FUNCTION_BLOCK FB_MotionVirtualFrame
(*
Takes 3 ST_MotionStages representing real axes that are orthogonal to each other and in a base frame of reference.
Takes 3 ST_MotionStages representing virtual axes that are orthogonal to each other and in a new frame of reference.
Computes the transformation from the base to the new frame of reference using 3 euler angles and a rotation order
as inputs. By default, the order and angles are interpreted as going from the base to the virtual frame. Can be
switched to go from virtual to base frame of reference.
If enabled, this function block will automatically handle commanding the real axes to move when the virtual axes
are commanded to move. If not enabled, the function block acts as a calculator, outputing the results of
calculating motions in a new frame of reference, but not changing any setpoints or commanding any moves.
*)
VAR_IN_OUT
    stMotionStageRx : ST_MotionStage; // Real X Axis in base frame of reference
    stMotionStageRy : ST_MotionStage; // Real Y Axis in base frame of reference
    stMotionStageRz : ST_MotionStage; // Real Z Axis in base frame of reference
    stMotionStageVx : ST_MotionStage; // Virtual X Axis in new frame of reference
    stMotionStageVy : ST_MotionStage; // Virtual Y Axis in new frame of reference
    stMotionStageVz : ST_MotionStage; // Virtual Z Axis in new frame of reference
END_VAR
VAR_INPUT
    (*TRUE to automatically overwrite real axis setpoints and command moves.
      FALSE to use this function only as a calculator.*)
    bEnable : BOOL;
    fAlphaDegrees : LREAL; // Angle of rotation about first axis.
    fBetaDegrees : LREAL; // Angle of rotation about second axis.
    fGammaDegrees : LREAL; // Angle of rotation about third axis.
    (*Rotation Order. E.g: XYZ to rotate alpha degrees around X axis, beta degrees around Y axis,
      and gamma degrees around Z axis. Valid rotation orders are:
      YZY, YXY, ZYZ, ZXZ, XYX, XZX, XYZ, YZX, ZXY, XZY, ZYX, YXZ.
      Default order for empty or invalid input is: ZYX.*)
    sOrder : STRING;
    (*FALSE to define inputs as rotating the frame of reference from the new frame to the base frame.
      TRUE to define the inputs as rotating the frame of reference from the base from to the new frame.*)
    bBaseToNew : BOOL := TRUE;
END_VAR
VAR_OUTPUT
    fbVirtActPositionVec3 : FB_Vec3;
    fbVirtActVelocityVec3 : FB_Vec3;
    fbVirtActAcceleraVec3 : FB_Vec3;

    fbRealTarPositionVec3 : FB_Vec3;
    fbRealTarVelocityVec3 : FB_Vec3;
    fbRealTarAcceleraVec3 : FB_Vec3;
END_VAR
VAR
    fAlphaRadians : LREAL;
    fBetaRadians : LREAL;
    fGammaRadians : LREAL;

    rtExecuteVx : R_TRIG;
    rtExecuteVy : R_TRIG;
    rtExecuteVz : R_TRIG;

    fbRealActPositionVec3 : FB_Vec3;
    fbRealActVelocityVec3 : FB_Vec3;
    fbRealActAcceleraVec3 : FB_Vec3;

    sOrderReversed : STRING;
    sLeft : STRING;
    sMid : STRING;
    sRight : STRING;

    fbVirtTarPositionVec3 : FB_Vec3;
    fbVirtTarVelocityVec3 : FB_Vec3;
    fbVirtTarAcceleraVec3 : FB_Vec3;
END_VAR


fAlphaRadians := DegToRad(fAlphaDegrees);
fBetaRadians := DegToRad(fBetaDegrees);
fGammaRadians := DegToRad(fGammaDegrees);

rtExecuteVx(CLK := stMotionStageVx.bExecute);
rtExecuteVy(CLK := stMotionStageVy.bExecute);
rtExecuteVz(CLK := stMotionStageVz.bExecute);

fbRealActPositionVec3.x := stMotionStageRx.Axis.NcToPlc.ActPos;
fbRealActPositionVec3.y := stMotionStageRy.Axis.NcToPlc.ActPos;
fbRealActPositionVec3.z := stMotionStageRz.Axis.NcToPlc.ActPos;

fbRealActVelocityVec3.x := stMotionStageRx.Axis.NcToPlc.ActVelo;
fbRealActVelocityVec3.y := stMotionStageRy.Axis.NcToPlc.ActVelo;
fbRealActVelocityVec3.z := stMotionStageRz.Axis.NcToPlc.ActVelo;

fbRealActAcceleraVec3.x := stMotionStageRx.Axis.NcToPlc.ActAcc;
fbRealActAcceleraVec3.y := stMotionStageRy.Axis.NcToPlc.ActAcc;
fbRealActAcceleraVec3.z := stMotionStageRz.Axis.NcToPlc.ActAcc;

sOrderReversed := ReverseOrder(sOrder);

IF bBaseToNew THEN
    RotatePosVelAccFrame(
        fbBaseFramePositionVec3 := fbRealActPositionVec3,
        fbBaseFrameVelocityVec3 := fbRealActVelocityVec3,
        fbBaseFrameAcceleraVec3 := fbRealActAcceleraVec3,
        fbNewFramePositionVec3 => fbVirtActPositionVec3,
        fbNewFrameVelocityVec3 => fbVirtActVelocityVec3,
        fbNewFrameAcceleraVec3 => fbVirtActAcceleraVec3,
        fAlphaRadians := fAlphaRadians,
        fBetaRadians := fBetaRadians,
        fGammaRadians := fGammaRadians,
        sOrder := sOrder
    );
ELSE
    RotatePosVelAccFrame(
        fbBaseFramePositionVec3 := fbRealActPositionVec3,
        fbBaseFrameVelocityVec3 := fbRealActVelocityVec3,
        fbBaseFrameAcceleraVec3 := fbRealActAcceleraVec3,
        fbNewFramePositionVec3 => fbVirtActPositionVec3,
        fbNewFrameVelocityVec3 => fbVirtActVelocityVec3,
        fbNewFrameAcceleraVec3 => fbVirtActAcceleraVec3,
        fAlphaRadians := -fGammaRadians,
        fBetaRadians := -fBetaRadians,
        fGammaRadians := -fAlphaRadians,
        sOrder := sOrderReversed
    );
END_IF

SetTargetPosVelAcc3D(
    stMotionStageX := stMotionStageVx,
    stMotionStageY := stMotionStageVy,
    stMotionStageZ := stMotionStageVz,
    fbActPosVec3 := fbVirtActPositionVec3,
    fbTarPosVec3 => fbVirtTarPositionVec3,
    fbTarVelVec3 => fbVirtTarVelocityVec3,
    fbTarAccVec3 => fbVirtTarAcceleraVec3
);

IF bBaseToNew THEN
    RotatePosVelAccFrame(
        fbBaseFramePositionVec3 := fbVirtTarPositionVec3,
        fbBaseFrameVelocityVec3 := fbVirtTarVelocityVec3,
        fbBaseFrameAcceleraVec3 := fbVirtTarAcceleraVec3,
        fbNewFramePositionVec3 => fbRealTarPositionVec3,
        fbNewFrameVelocityVec3 => fbRealTarVelocityVec3,
        fbNewFrameAcceleraVec3 => fbRealTarAcceleraVec3,
        fAlphaRadians := -fGammaRadians,
        fBetaRadians := -fBetaRadians,
        fGammaRadians := -fAlphaRadians,
        sOrder := sOrderReversed
    );
ELSE
    RotatePosVelAccFrame(
        fbBaseFramePositionVec3 := fbVirtTarPositionVec3,
        fbBaseFrameVelocityVec3 := fbVirtTarVelocityVec3,
        fbBaseFrameAcceleraVec3 := fbVirtTarAcceleraVec3,
        fbNewFramePositionVec3 => fbRealTarPositionVec3,
        fbNewFrameVelocityVec3 => fbRealTarVelocityVec3,
        fbNewFrameAcceleraVec3 => fbRealTarAcceleraVec3,
        fAlphaRadians := fAlphaRadians,
        fBetaRadians := fBetaRadians,
        fGammaRadians := fGammaRadians,
        sOrder := sOrder
    );
END_IF

IF bEnable THEN
    IF rtExecuteVx.Q OR rtExecuteVy.Q OR rtExecuteVz.Q THEN
        stMotionStageRx.fPosition := fbRealTarPositionVec3.x;
        stMotionStageRy.fPosition := fbRealTarPositionVec3.y;
        stMotionStageRz.fPosition := fbRealTarPositionVec3.z;

        stMotionStageRx.fVelocity := ABS(fbRealTarVelocityVec3.x);
        stMotionStageRy.fVelocity := ABS(fbRealTarVelocityVec3.y);
        stMotionStageRz.fVelocity := ABS(fbRealTarVelocityVec3.z);

        stMotionStageRx.fAcceleration := ABS(fbRealTarAcceleraVec3.x);
        stMotionStageRy.fAcceleration := ABS(fbRealTarAcceleraVec3.y);
        stMotionStageRz.fAcceleration := ABS(fbRealTarAcceleraVec3.z);

        stMotionStageRx.fDeceleration := ABS(fbRealTarAcceleraVec3.x);
        stMotionStageRy.fDeceleration := ABS(fbRealTarAcceleraVec3.y);
        stMotionStageRz.fDeceleration := ABS(fbRealTarAcceleraVec3.z);

        IF stMotionStageRx.fVelocity >= 0.001 THEN
            stMotionStageRx.bMoveCmd := TRUE;
        ELSIF ABS(stMotionStageRx.fPosition - stMotionStageRx.Axis.NcToPlc.ActPos) >
                stMotionStageRx.stAxisParameters.fTargetPosControlRange THEN
            stMotionStageRx.fVelocity := 0.001;
            stMotionStageRx.bMoveCmd := TRUE;
        END_IF

        IF stMotionStageRy.fVelocity >= 0.001 THEN
            stMotionStageRy.bMoveCmd := TRUE;
        ELSIF ABS(stMotionStageRy.fPosition - stMotionStageRy.Axis.NcToPlc.ActPos) >
                stMotionStageRy.stAxisParameters.fTargetPosControlRange THEN
            stMotionStageRy.fVelocity := 0.001;
            stMotionStageRy.bMoveCmd := TRUE;
        END_IF

        IF stMotionStageRz.fVelocity >= 0.001 THEN
            stMotionStageRz.bMoveCmd := TRUE;
        ELSIF ABS(stMotionStageRz.fPosition - stMotionStageRz.Axis.NcToPlc.ActPos) >
                stMotionStageRz.stAxisParameters.fTargetPosControlRange THEN
            stMotionStageRz.fVelocity := 0.001;
            stMotionStageRz.bMoveCmd := TRUE;
        END_IF
    END_IF

    IF stMotionStageRx.bError OR stMotionStageRy.bError OR stMotionStageRz.bError THEN
        stMotionStageVx.bError := TRUE;
        stMotionStageVy.bError := TRUE;
        stMotionStageVz.bError := TRUE;
        stMotionStageVx.sCustomErrorMessage := 'An error occured in one of the real axes. All virtual axes stopped.';
        stMotionStageVy.sCustomErrorMessage := 'An error occured in one of the real axes. All virtual axes stopped.';
        stMotionStageVz.sCustomErrorMessage := 'An error occured in one of the real axes. All virtual axes stopped.';
    END_IF
END_IF


METHOD PUBLIC DegToRad : LREAL
VAR_INPUT
    fDeg : LREAL;
END_VAR

DegToRad := fDeg  / 180.0 * lcls_twincat_math.GVL_Constants.PI;
END_METHOD

METHOD ReverseOrder : STRING
VAR_INPUT
    sOrder : STRING;
END_VAR

IF sOrder = '' THEN
    sOrder := 'ZYX';
END_IF
sLeft := LEFT(sOrder, 1);
sMid := MID(sOrder, 2, 1);
sRight := RIGHT(sOrder, 1);
ReverseOrder := CONCAT(sRight, CONCAT(sMid, sLeft));
END_METHOD


METHOD PUBLIC RotatePosVelAccFrame
VAR_INPUT
    fbBaseFramePositionVec3 : FB_Vec3;
    fbBaseFrameVelocityVec3 : FB_Vec3;
    fbBaseFrameAcceleraVec3 : FB_Vec3;

    fAlphaRadians : LREAL;
    fBetaRadians : LREAL;
    fGammaRadians : LREAL;
    sOrder : STRING;
END_VAR
VAR_OUTPUT
    fbNewFramePositionVec3 : FB_Vec3;
    fbNewFrameVelocityVec3 : FB_Vec3;
    fbNewFrameAcceleraVec3 : FB_Vec3;
END_VAR

fbNewFramePositionVec3 := F_EulerRotateVec3Frame(
    iVec3 := fbBaseFramePositionVec3,
    fAlphaRadians := fAlphaRadians,
    fBetaRadians := fBetaRadians,
    fGammaRadians := fGammaRadians,
    sOrder := sOrder
);

fbNewFrameVelocityVec3 := F_EulerRotateVec3Frame(
    iVec3 := fbBaseFrameVelocityVec3,
    fAlphaRadians := fAlphaRadians,
    fBetaRadians := fBetaRadians,
    fGammaRadians := fGammaRadians,
    sOrder := sOrder
);

fbNewFrameAcceleraVec3 := F_EulerRotateVec3Frame(
    iVec3 := fbBaseFrameAcceleraVec3,
    fAlphaRadians := fAlphaRadians,
    fBetaRadians := fBetaRadians,
    fGammaRadians := fGammaRadians,
    sOrder := sOrder
);
END_METHOD


METHOD PUBLIC SetTargetPosVelAcc1D
VAR_INPUT
    stMotionStage : ST_MotionStage;
    fActPos : LREAL;
END_VAR
VAR_OUTPUT
    fTarPos : LREAL;
    fTarVel : LREAL;
    fTarAcc : LREAL;
END_VAR

IF stMotionStage.bBusy THEN
    fTarPos := stMotionStage.fPosition;
    IF fTarPos >= fActPos THEN
        fTarVel := stMotionStage.fVelocity;
        fTarAcc := stMotionStage.fAcceleration;
    ELSE
        fTarVel := -stMotionStage.fVelocity;
        fTarAcc := -stMotionStage.fAcceleration;
    END_IF
ELSE
    fTarPos := fActPos;
    fTarVel := 0.0;
    fTarAcc := 0.0;
END_IF
END_METHOD


METHOD PUBLIC SetTargetPosVelAcc3D
VAR_INPUT
    stMotionStageX : ST_MotionStage;
    stMotionStageY : ST_MotionStage;
    stMotionStageZ : ST_MotionStage;
    fbActPosVec3 : FB_Vec3;
END_VAR
VAR_OUTPUT
    fbTarPosVec3 : FB_Vec3;
    fbTarVelVec3 : FB_Vec3;
    fbTarAccVec3 : FB_Vec3;
END_VAR
VAR
    fTarPosX : LREAL;
    fTarPosY : LREAL;
    fTarPosZ : LREAL;

    fTarVelX : LREAL;
    fTarVelY : LREAL;
    fTarVelZ : LREAL;

    fTarAccX : LREAL;
    fTarAccY : LREAL;
    fTarAccZ : LREAL;
END_VAR

SetTargetPosVelAcc1D(
    stMotionStage := stMotionStageX,
    fActPos := fbActPosVec3.x,
    fTarPos => fTarPosX,
    fTarVel => fTarVelX,
    fTarAcc => fTarAccX
);

SetTargetPosVelAcc1D(
    stMotionStage := stMotionStageY,
    fActPos := fbActPosVec3.y,
    fTarPos => fTarPosY,
    fTarVel => fTarVelY,
    fTarAcc => fTarAccY
);

SetTargetPosVelAcc1D(
    stMotionStage := stMotionStageZ,
    fActPos := fbActPosVec3.z,
    fTarPos => fTarPosZ,
    fTarVel => fTarVelZ,
    fTarAcc => fTarAccZ
);

fbTarPosVec3.Set(fTarPosX, fTarPosY, fTarPosZ);
fbTarVelVec3.Set(fTarVelX, fTarVelY, fTarVelZ);
fbTarAccVec3.Set(fTarAccX, fTarAccY, fTarAccZ);
END_METHOD

END_FUNCTION_BLOCK

(* stored: Version 1.1.0.1, ProductVersion 3.1.4022.18
   POU FB_MotionVirtualFrame: Id {db4a3323-bc78-4bca-8918-99f0e2117f18}, SpecialFunc None
   Method DegToRad: Id {b3994cfb-0e95-49f7-8a93-c949b8827612}
   Method ReverseOrder: Id {ad0bf132-fcf3-412d-9abf-164f39420901}
   Method RotatePosVelAccFrame: Id {61c7d3bf-c97e-4994-9217-9ace0f7272b1}
   Method SetTargetPosVelAcc1D: Id {c0957557-35ec-4203-a92e-41f437a57b08}
   Method SetTargetPosVelAcc3D: Id {7ca16bbb-14b2-4a45-b834-72e712c8fe8d} *)
